FUNCTION_BLOCK Test_GetTestHandlesInvalidIndex EXTENDS T_UnitTestBase
VAR
    List : T_ListOfTests(Capacity := 10);
END_VAR

METHOD Init
List.Clear();
END_METHOD

PROPERTY Name : Tc2_System.T_MaxString
GET
END_GET
END_PROPERTY

METHOD RunTest
VAR_OUTPUT
    TestCompleted : BOOL;
    TestFailed    : BOOL;
END_VAR
VAR_INST
    TestNumber4 : I_UnitTest;
END_VAR
TestNumber4 := List.GetTest(4);

AssertTrue(Source    := TestName,
             Condition := (TestNumber4 = 0),
             Message   := 'GetTest() has unexpected return value',
             Failed    => TestFailed);

TestCompleted := TRUE;
END_METHOD

END_FUNCTION_BLOCK

(* stored: Version 1.1.0.1, ProductVersion 3.1.4024.12
   POU Test_GetTestHandlesInvalidIndex: Id {f2759aac-dc6b-41e7-b261-e0a7bb0a9059}, SpecialFunc None
   Method Init: Id {0089e835-1319-41ef-a4d8-adb3b99d0a47}
   Property Name: Id {4a77067e-3885-4fc4-8152-205388f90c47}
   Get Get: Id {278475f0-5263-4538-82fd-fa1afe6878db}
   Method RunTest: Id {196a1154-4f83-4db1-bc9d-8909993894ea} *)
